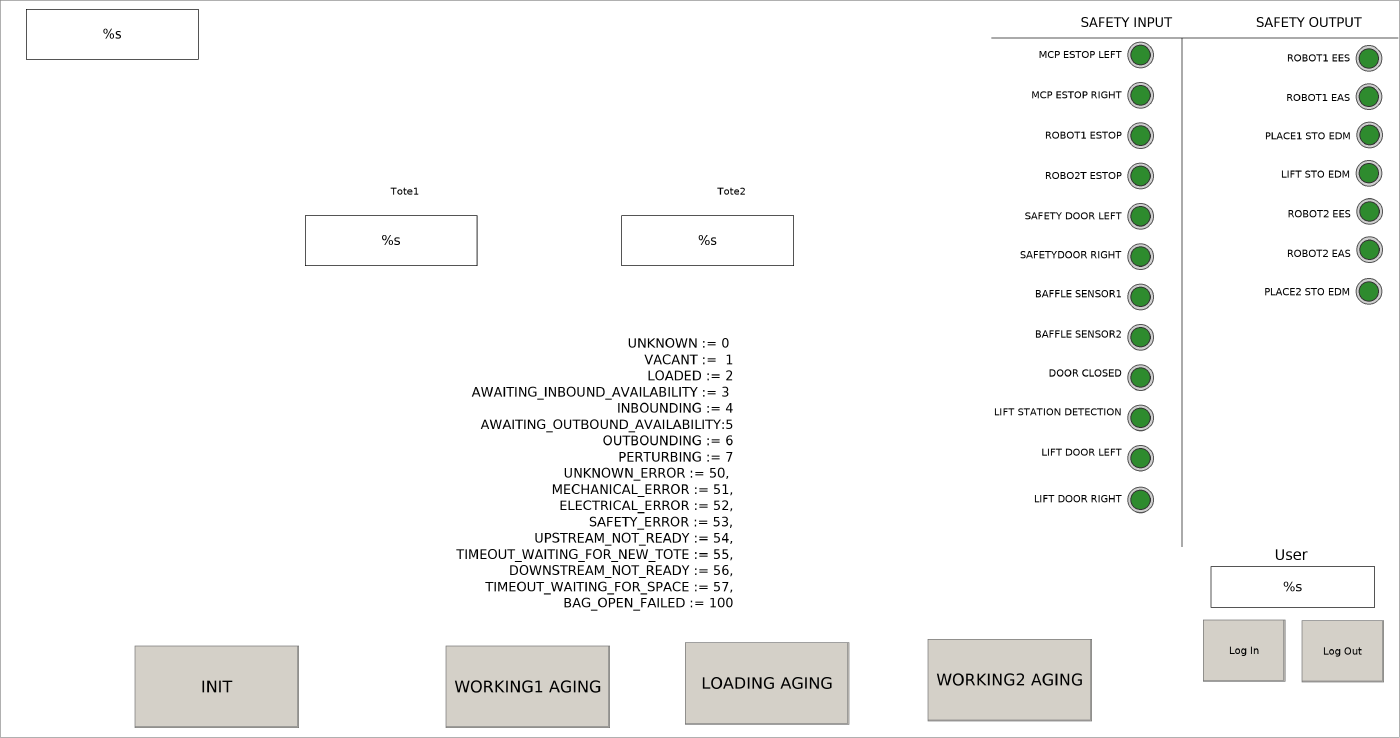
VISUALIZATION visu_operation  // 2048x1080
    Button (197,945 240x120), "INIT", colour toggle: G_HMI.bInit
        OnMouseDown: execute { G_HMI.bInit	:= TRUE; }
        OnMouseUp: execute { G_HMI.bInit	:= FALSE; }
    Lamp1 (1646,58 45x45), variable: MAIN.safety_1.mcp_estop_left.Q, style: Lamp-Lamp1-Green
    Label (1344,65 300x30), "MCP ESTOP LEFT"
    Lamp1 (1646,117 45x45), variable: MAIN.safety_1.mcp_estop_right.Q, style: Lamp-Lamp1-Green
    Label (1344,124 300x30), "MCP ESTOP RIGHT"
    Lamp1 (1646,353 45x45), variable: MAIN.safety_1.safetyDoor_right, style: Lamp-Lamp1-Green
    Label (1344,360 300x26), "SAFETYDOOR RIGHT"
    Lamp1 (1646,530 45x45), variable: MAIN.safety_1.door_closed, style: Lamp-Lamp1-Green
    Label (1344,533 300x26), "DOOR CLOSED"
    Lamp1 (1646,589 45x45), variable: MAIN.safety_1.lift_station_detection, style: Lamp-Lamp1-Green
    Label (1344,588 300x30), "LIFT STATION DETECTION"
    Lamp1 (1980,63 45x45), variable: GVL_SAFETY.robot1_STO_EES, style: Lamp-Lamp1-Green
    Label (1728,70 250x30), "ROBOT1 EES"
    Lamp1 (1980,231 45x45), variable: GVL_SAFETY.Lift_STO, style: Lamp-Lamp1-Green
    Label (1728,240 250x30), "LIFT STO EDM"
    Lamp1 (1981,175 45x45), variable: GVL_SAFETY.Place1_STO, style: Lamp-Lamp1-Green
    Label (1729,186 250x26), "PLACE1 STO EDM"
    Lamp1 (1980,404 45x45), variable: GVL_SAFETY.Place2_STO, style: Lamp-Lamp1-Green
    Label (1728,414 250x26), "PLACE2 STO EDM"
    Lamp1 (1980,119 45x45), variable: GVL_SAFETY.robot1_STO_EAS, style: Lamp-Lamp1-Green
    Label (1728,128 250x30), "ROBOT1 EAS"
    Line (1729,800) (1729,55)
    Label (1523,18 250x30), "SAFETY INPUT"
    Label (1790,18 250x30), "SAFETY OUTPUT"
    Line (1450,55) (2045,55)
    Rectangle (38,13 252x74), "%s"
    Rectangle (1771,829 240x60), "%s", text variable: G_HMI.sLoginnedUser
    Button (1904,908 120x90), "Log Out"
        OnMouseDown: VisuUserMgmt Type=Logout
    Button (1760,907 120x90), "Log In"
        OnMouseDown: VisuUserMgmt Type=Login
    Label (1814,797 150x30), "User"
    Label (1344,647 300x30), "LIFT DOOR LEFT"
    Lamp1 (1646,648 45x45), variable: MAIN.safety_1.lift_door_left.Q, style: Lamp-Lamp1-Green
    Label (1344,715 300x30), "LIFT DOOR RIGHT"
    Lamp1 (1646,709 45x45), variable: MAIN.safety_1.lift_door_right.Q, style: Lamp-Lamp1-Green
    Label (1344,301 300x30), "SAFETY DOOR LEFT"
    Lamp1 (1646,294 45x45), variable: MAIN.safety_1.safetyDoor_left, style: Lamp-Lamp1-Green
    Label (1344,415 300x30), "BAFFLE SENSOR1"
    Lamp1 (1646,412 45x45), variable: MAIN.safety_1.baffle_sensor_1, style: Lamp-Lamp1-Green
    Label (1344,474 300x30), "BAFFLE SENSOR2"
    Lamp1 (1646,471 45x45), variable: MAIN.safety_1.baffle_sensor_2, style: Lamp-Lamp1-Green
    Lamp1 (1981,287 45x45), variable: GVL_SAFETY.robot2_STO_EES, style: Lamp-Lamp1-Green
    Label (1729,298 250x30), "ROBOT2 EES"
    Lamp1 (1981,343 45x45), variable: GVL_SAFETY.robot2_STO_EAS, style: Lamp-Lamp1-Green
    Label (1729,356 250x30), "ROBOT2 EAS"
    Lamp1 (1646,176 45x45), variable: MAIN.safety_1.bRobot1_eStop, style: Lamp-Lamp1-Green
    Label (1344,183 300x30), "ROBOT1 ESTOP"
    Lamp1 (1646,235 45x45), variable: MAIN.safety_1.bRobot2_eStop, style: Lamp-Lamp1-Green
    Label (1344,242 300x30), "ROBO2T ESTOP"
    Label (316,265 300x30), "Tote1"
    Rectangle (446,315 252x74), "%s", text variable: GVL.fb_working1.tote_status
    Label (314,457 762x471), "UNKNOWN := 0 VACANT := 1 LOADED := 2 AWAITING_INBOUND_AVAILABILITY := 3 INBOUNDING := 4 AWAITING_OUTBOUND_AVAILABILITY:5 OUTBOUNDING := 6 PERTURBING := 7 UNKNOWN_ERROR := 50, MECHANICAL_ERROR := 51, ELECTRICAL_ERROR := 52, SAFETY_ERROR := 53, UPSTREAM_NOT_READY := 54, TIMEOUT_WAITING_FOR_NEW_TOTE := 55, DOWNSTREAM_NOT_READY := 56, TIMEOUT_WAITING_FOR_SPACE := 57, BAG_OPEN_FAILED := 100"
    Rectangle (909,315 252x74), "%s", text variable: GVL.fb_working2.tote_status
    Label (794,265 300x30), "Tote2"
    Button (652,945 240x120), "WORKING1 AGING"
        toggle GVL.fb_working1.bAging_test
    Button (1002,940 240x120), "LOADING AGING"
        toggle GVL.fb_loading.bAging_test
    Button (1357,935 240x120), "WORKING2 AGING"
        toggle GVL.fb_working2.bAging_test
END_VISUALIZATION

(* stored: Version 1.1.0.1, ProductVersion 3.1.4024.12
   Visu visu_operation: Id {4abbf3f6-c173-4bcb-82b6-c0f3163ef68d} *)
